# EPICS substitutions: backup/mc11/tpmacApp/Db/motorstatus.substitutions
file "db/motorstatus.db"
{
pattern
{SYS,              DEV,                 PORT,  AXIS }
{"XF:23ID1-ES",  "{Dif:Tbl-Ax:Z1}",        "P0",   1   }
{"XF:23ID1-ES",  "{Dif:Tbl-Ax:Z2}",        "P0",   2   }
{"XF:23ID1-ES",  "{Dif:Tbl-Ax:Z3}",        "P0",   3   }
{"XF:23ID1-ES",  "{Dif:Tbl-Ax:X1}",        "P0",   4   }
{"XF:23ID1-ES",  "{Dif:Tbl-Ax:X2}",        "P0",   5   }

}

file "db/pmacStatusAxis.db"
{
pattern
{SYS,               DEV,           PORT,  AXIS }
{"XF:23ID1-CT",  "{MC:11-Ax:1}",   "P0",   1   }
{"XF:23ID1-CT",  "{MC:11-Ax:2}",   "P0",   2   }
{"XF:23ID1-CT",  "{MC:11-Ax:3}",   "P0",   3   }
{"XF:23ID1-CT",  "{MC:11-Ax:4}",   "P0",   4   }
{"XF:23ID1-CT",  "{MC:11-Ax:5}",   "P0",   5   }

}
